(* Logix 5000 project; controller VET 1756-L62 rev 19.52; software revision 19.01; part 12 of 27 *)
(* tags used below, declared in another part *)
   bufferF : REAL[5];
   dosif_struct : ALIAS FOR dosificador[0];
   dosificacion_interrumpida : BOOL;
   dosificando : BOOL;
   falla_struct : falla_aux;
   flags : DINT;
   frq : ALIAS FOR dosif_struct.frq_terreno;
   frq_calculada : REAL;
   idx_batch : DINT;
   idx_bin : DINT;
   idx_ing : DINT;
   idx_tabbin : DINT;
   idx_tolv : DINT;   // Índice de Tolva
   limite_err_inf : REAL;
   limite_err_sup : REAL;
   mensaje : ALIAS FOR dosif_struct.msg;
   peso_delta : REAL;
   peso_detencion : REAL;
   peso_max : REAL;
   peso_medido : ALIAS FOR dosif_struct.peso_terreno;
   peso_neto : REAL;
   peso_objetivo : REAL;
   precorte : REAL;
   respuesta : ALIAS FOR dosif_struct.ans;
   resultado : ALIAS FOR dosif_struct.resultado;
   setD : DINT[5];
   setF : REAL[5];
   step_index : DINT;
   step_index_buffer : DINT;
   T : TIMER[15];
   t_espera : DINT;
   t_pulso : DINT;
   tara : REAL;
   _Eqp : Equipo[800];
   Batch : batch[10];
   Dosificar_MAC_01 : PHASE;
   fecha_plc : DINT;
   hora_plc : DINT;
   TabBin : Bins_Setup;
(* Dosificar_MAC_01, continued *)

ROUTINE dosificar   (* ladder *)
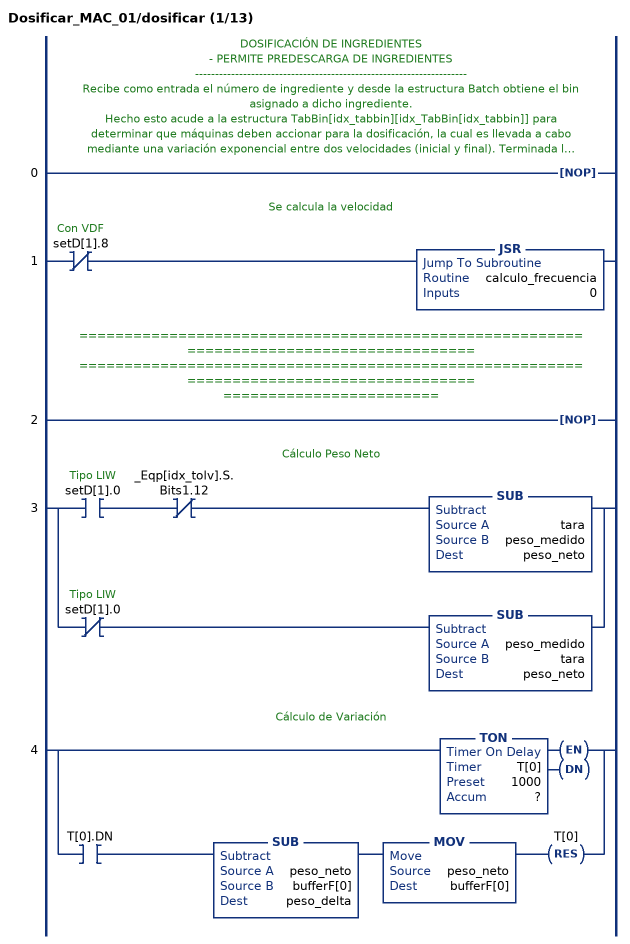
   // DOSIFICACIÓN DE INGREDIENTES
   // - PERMITE PREDESCARGA DE INGREDIENTES
   // --------------------------------------------------------------------
   // Recibe como entrada el número de ingrediente y desde la estructura Batch obtiene el bin asignado a dicho ingrediente.
   // Hecho esto acude a la estructura TabBin[idx_tabbin][idx_TabBin[idx_tabbin]] para determinar que máquinas deben accionar para la dosificación, la cual es llevada a cabo
   // mediante una variación exponencial entre dos velocidades (inicial y final). Terminada la dosificación, se retornan o consolidan los aprendizajes
   // prBatchios de la dosificación, reflejados en un precorte ajustado.
   0: NOP();
   // Se calcula la velocidad
   1: XIO(setD[1].8)JSR(calculo_frecuencia,0);
   // ========================================================================================
   // ========================================================================================
   // ========================
   2: NOP();
   // Cálculo Peso Neto
   3: [XIC(setD[1].0) XIO(_Eqp[idx_tolv].S.Bits1.12) SUB(tara,peso_medido,peso_neto) ,XIO(setD[1].0) SUB(peso_medido,tara,peso_neto) ];
   // Cálculo de Variación
   4: [TON(T[0],?,?) ,XIC(T[0].DN) SUB(peso_neto,bufferF[0],peso_delta) MOV(peso_neto,bufferF[0]) RES(T[0]) ];
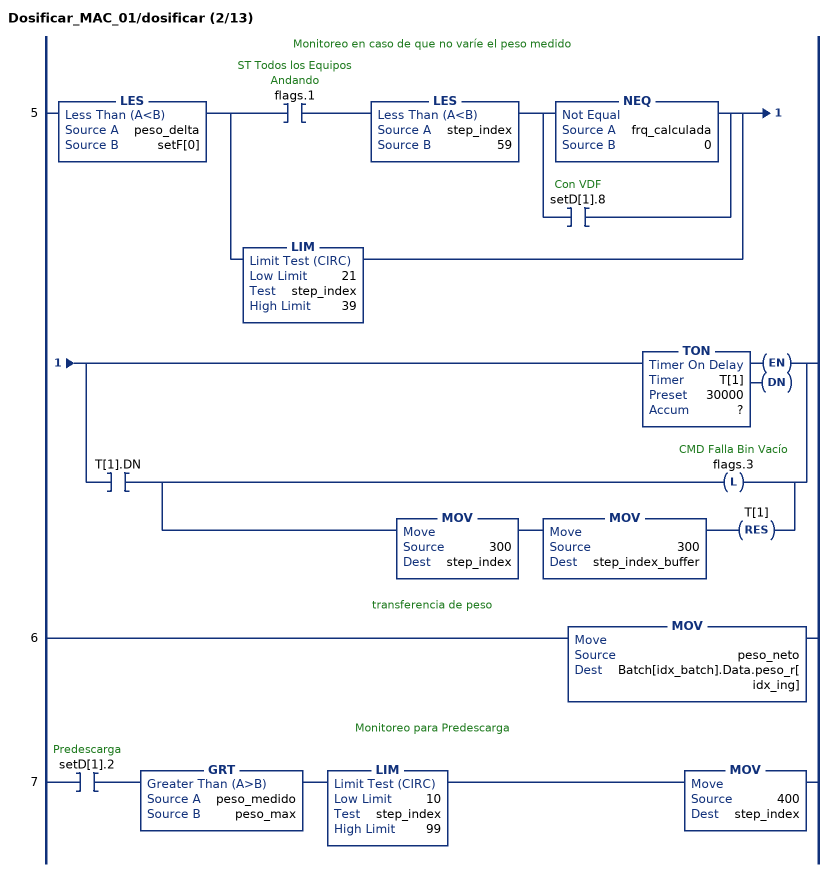
   // Monitoreo en caso de que no varíe el peso medido
   5: LES(peso_delta,setF[0])[XIC(flags.1) LES(step_index,59) [NEQ(frq_calculada,0) ,XIC(setD[1].8) ] ,LIM(21,step_index,39) ][TON(T[1],?,?) ,XIC(T[1].DN) [OTL(flags.3) ,MOV(300,step_index) MOV(300,step_index_buffer) RES(T[1]) ] ];
   // transferencia de peso
   6: MOV(peso_neto,Batch[idx_batch].Data.peso_r[idx_ing]);
   // Monitoreo para Predescarga
   7: XIC(setD[1].2)GRT(peso_medido,peso_max)LIM(10,step_index,99)MOV(400,step_index);
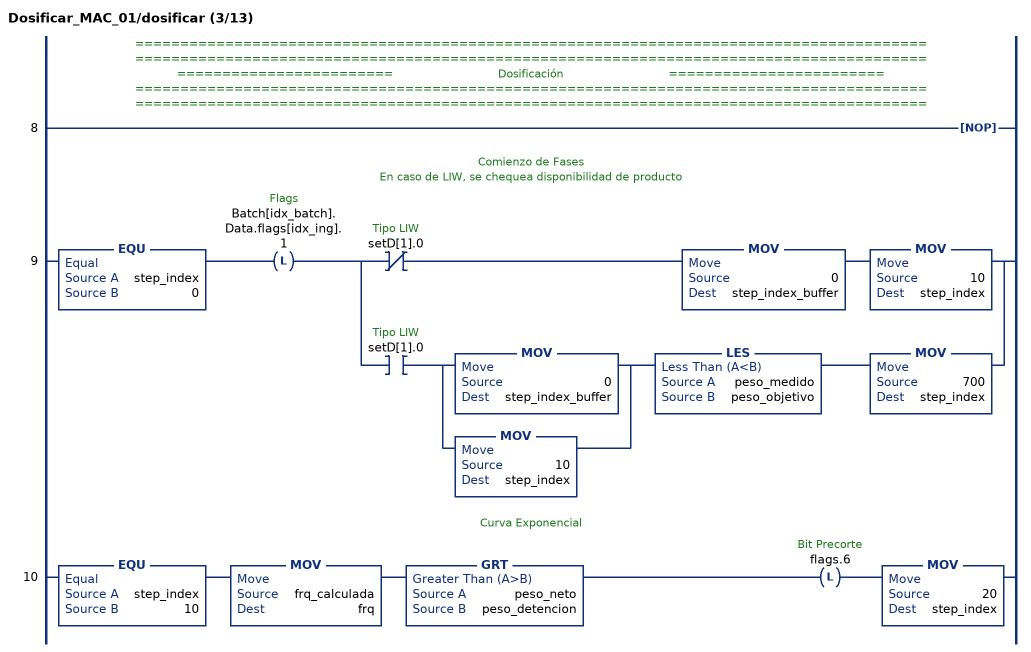
   // ========================================================================================
   // ========================================================================================
   // ========================                              Dosificación                              ========================
   // ========================================================================================
   // ========================================================================================
   8: NOP();
   // Comienzo de Fases
   // En caso de LIW, se chequea disponibilidad de producto
   9: EQU(step_index,0)OTL(Batch[idx_batch].Data.flags[idx_ing].1)[XIO(setD[1].0) MOV(0,step_index_buffer) MOV(10,step_index) ,XIC(setD[1].0) [MOV(0,step_index_buffer) ,MOV(10,step_index) ] LES(peso_medido,peso_objetivo) MOV(700,step_index) ];
   // Curva Exponencial
   10: EQU(step_index,10)MOV(frq_calculada,frq)GRT(peso_neto,peso_detencion)OTL(flags.6)MOV(20,step_index);
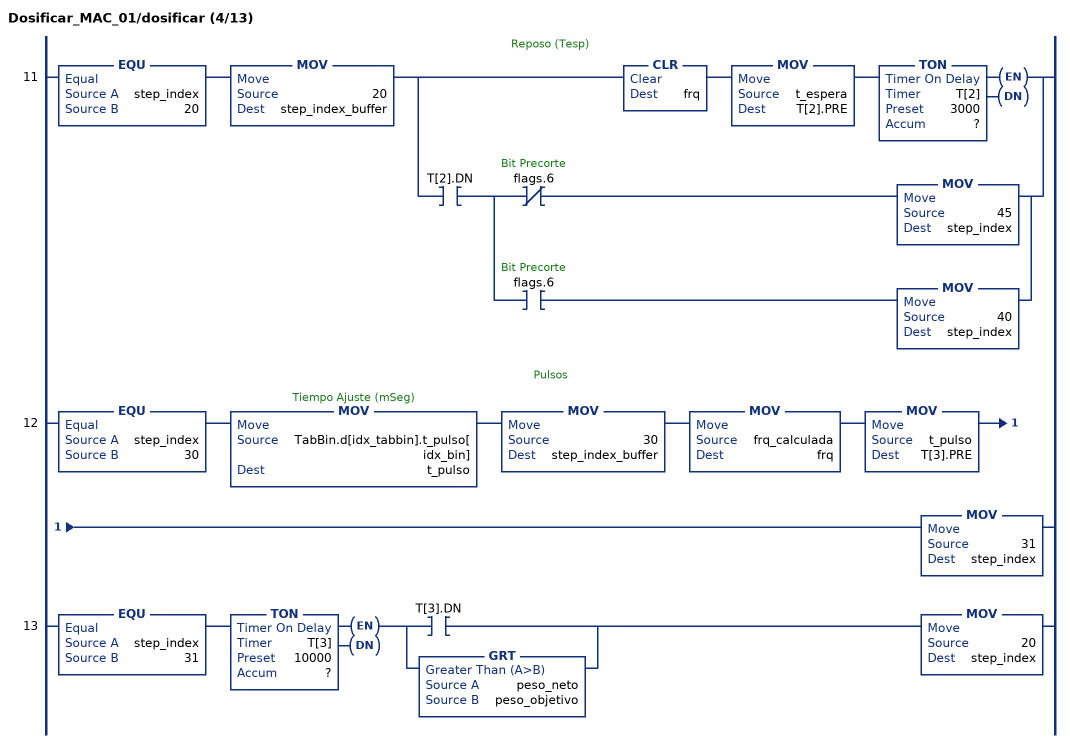
   // Reposo (Tesp)
   11: EQU(step_index,20)MOV(20,step_index_buffer)[CLR(frq) MOV(t_espera,T[2].PRE) TON(T[2],?,?) ,XIC(T[2].DN) [XIO(flags.6) MOV(45,step_index) ,XIC(flags.6) MOV(40,step_index) ] ];
   // Pulsos
   12: EQU(step_index,30)MOV(TabBin.d[idx_tabbin].t_pulso[idx_bin],t_pulso)MOV(30,step_index_buffer)MOV(frq_calculada,frq)MOV(t_pulso,T[3].PRE)MOV(31,step_index);
   13: EQU(step_index,31)TON(T[3],?,?)[XIC(T[3].DN) ,GRT(peso_neto,peso_objetivo) ]MOV(20,step_index);
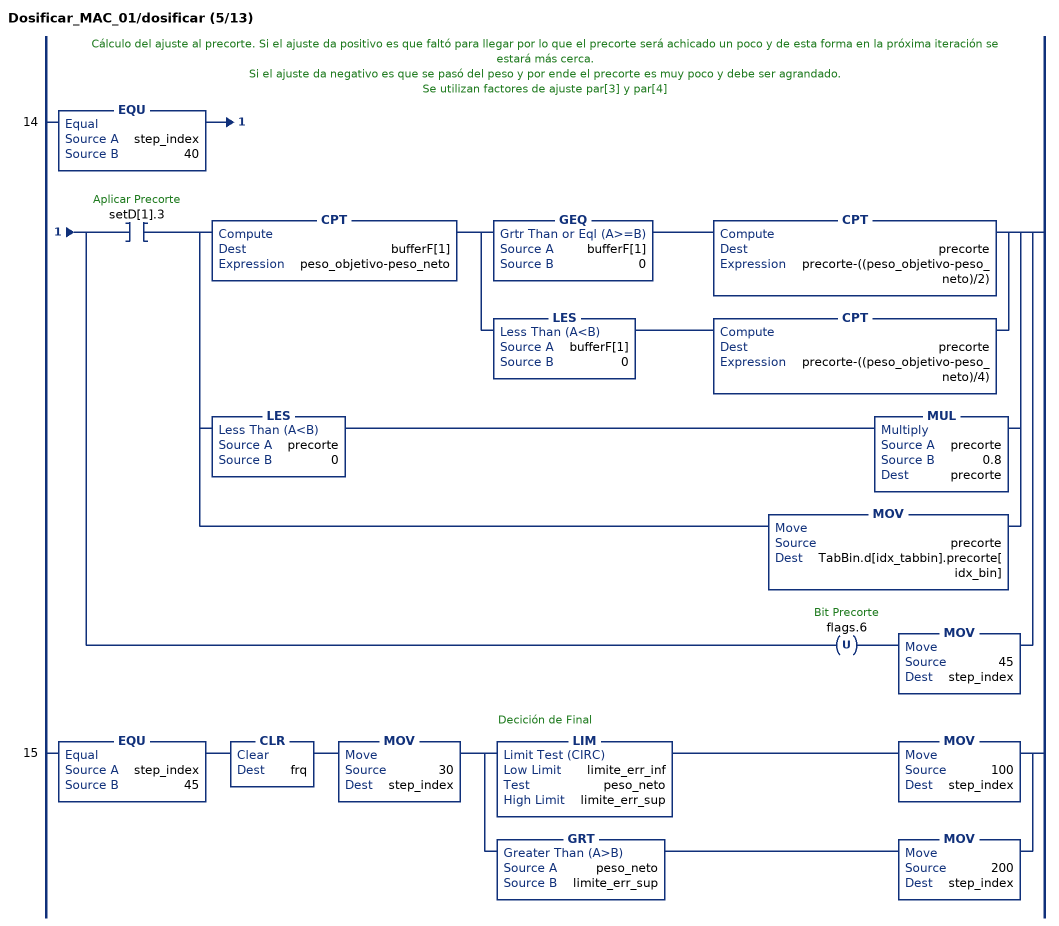
   // Cálculo del ajuste al precorte. Si el ajuste da positivo es que faltó para llegar por lo que el precorte será achicado un poco y de esta forma en la próxima iteración se estará más cerca.
   // Si el ajuste da negativo es que se pasó del peso y por ende el precorte es muy poco y debe ser agrandado.
   // Se utilizan factores de ajuste par[3] y par[4]
   14: EQU(step_index,40)[XIC(setD[1].3) [CPT(bufferF[1],peso_objetivo-peso_neto) [GEQ(bufferF[1],0) CPT(precorte,precorte-((peso_objetivo-peso_neto)/2)) ,LES(bufferF[1],0) CPT(precorte,precorte-((peso_objetivo-peso_neto)/4)) ] ,LES(precorte,0) MUL(precorte,0.8,precorte) ,MOV(precorte,TabBin.d[idx_tabbin].precorte[idx_bin]) ] ,OTU(flags.6) MOV(45,step_index) ];
   // Decición de Final
   15: EQU(step_index,45)CLR(frq)MOV(30,step_index)[LIM(limite_err_inf,peso_neto,limite_err_sup) MOV(100,step_index) ,GRT(peso_neto,limite_err_sup) MOV(200,step_index) ];
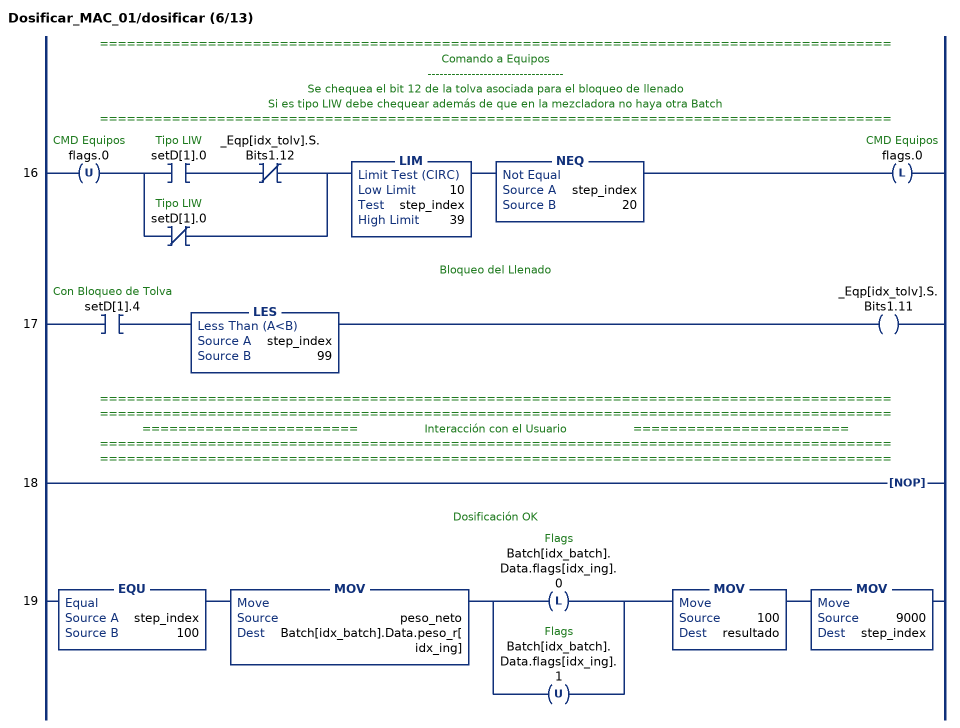
   // ========================================================================================
   // Comando a Equipos
   // ----------------------------------
   // Se chequea el bit 12 de la tolva asociada para el bloqueo de llenado
   // Si es tipo LIW debe chequear además de que en la mezcladora no haya otra Batch
   // ========================================================================================
   16: OTU(flags.0)[XIC(setD[1].0) XIO(_Eqp[idx_tolv].S.Bits1.12) ,XIO(setD[1].0) ]LIM(10,step_index,39)NEQ(step_index,20)OTL(flags.0);
   // Bloqueo del Llenado
   17: XIC(setD[1].4)LES(step_index,99)OTE(_Eqp[idx_tolv].S.Bits1.11);
   // ========================================================================================
   // ========================================================================================
   // ========================                   Interacción con el Usuario                   ========================
   // ========================================================================================
   // ========================================================================================
   18: NOP();
   // Dosificación OK
   19: EQU(step_index,100)MOV(peso_neto,Batch[idx_batch].Data.peso_r[idx_ing])[OTL(Batch[idx_batch].Data.flags[idx_ing].0) ,OTU(Batch[idx_batch].Data.flags[idx_ing].1) ]MOV(100,resultado)MOV(9000,step_index);
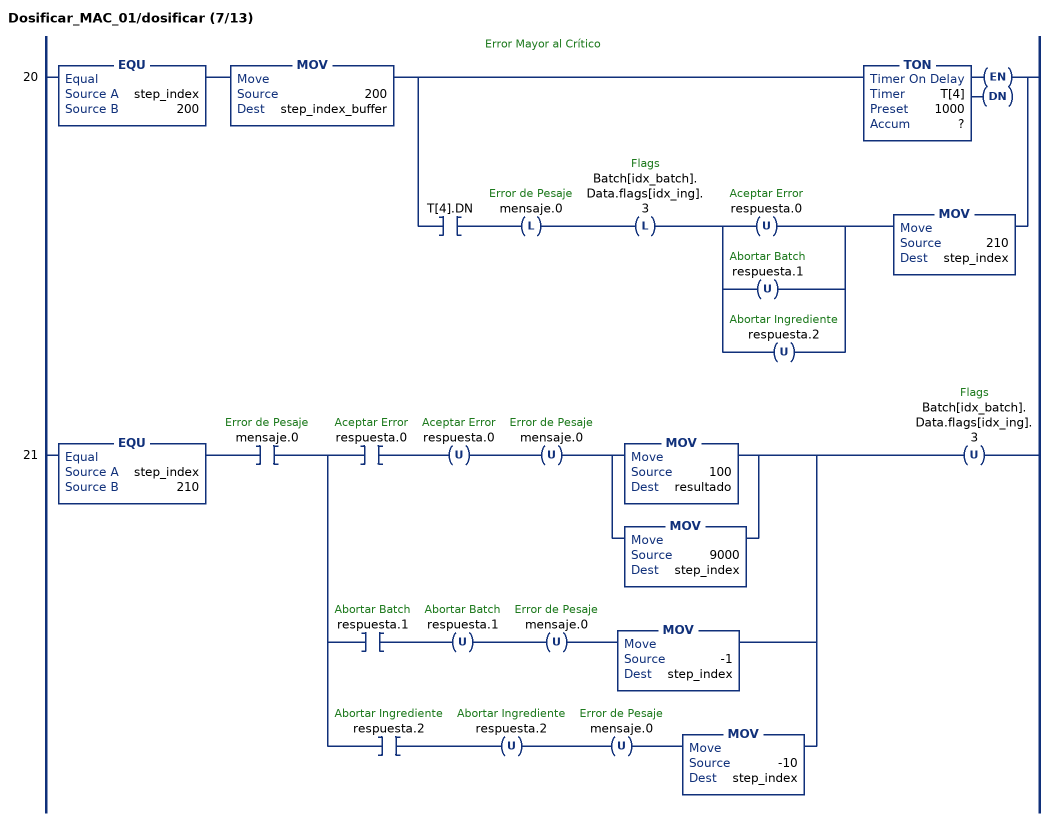
   // Error Mayor al Crítico
   20: EQU(step_index,200)MOV(200,step_index_buffer)[TON(T[4],?,?) ,XIC(T[4].DN) OTL(mensaje.0) OTL(Batch[idx_batch].Data.flags[idx_ing].3) [OTU(respuesta.0) ,OTU(respuesta.1) ,OTU(respuesta.2) ] MOV(210,step_index) ];
   21: EQU(step_index,210)XIC(mensaje.0)[XIC(respuesta.0) OTU(respuesta.0) OTU(mensaje.0) [MOV(100,resultado) ,MOV(9000,step_index) ] ,XIC(respuesta.1) OTU(respuesta.1) OTU(mensaje.0) MOV(-1,step_index) ,XIC(respuesta.2) OTU(respuesta.2) OTU(mensaje.0) MOV(-10,step_index) ]OTU(Batch[idx_batch].Data.flags[idx_ing].3);
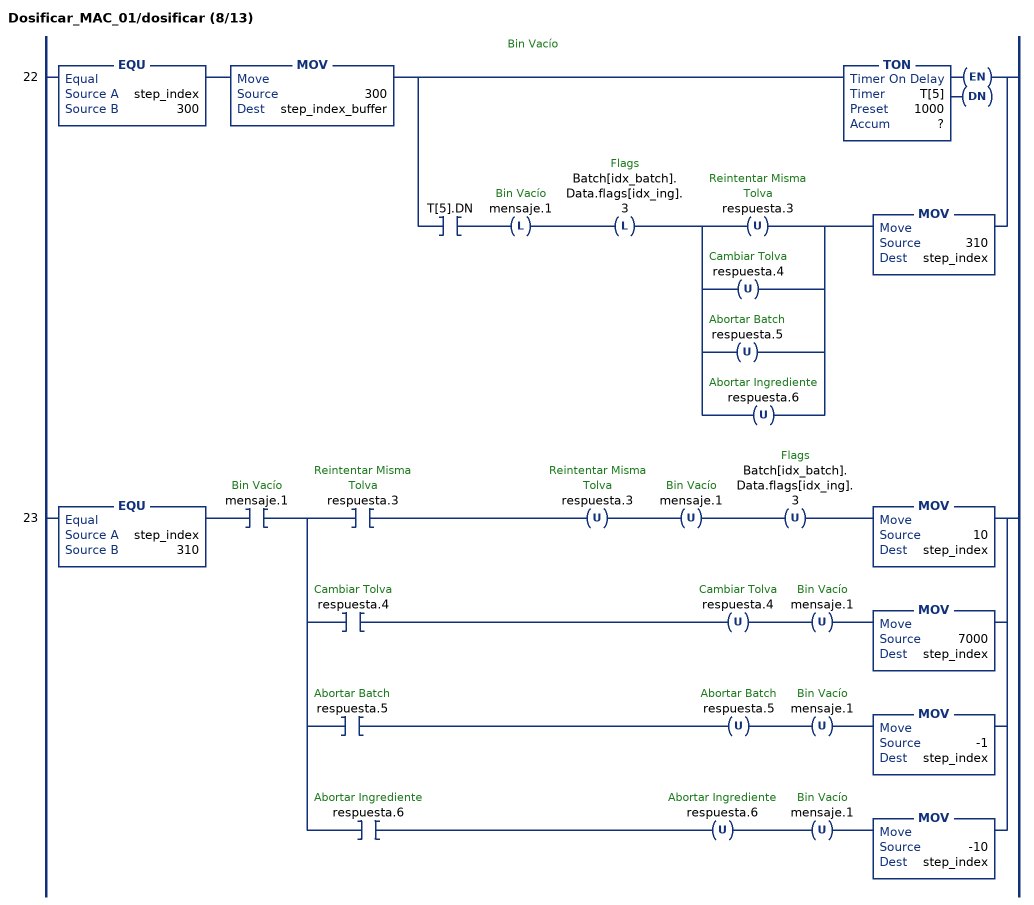
   // Bin Vacío
   22: EQU(step_index,300)MOV(300,step_index_buffer)[TON(T[5],?,?) ,XIC(T[5].DN) OTL(mensaje.1) OTL(Batch[idx_batch].Data.flags[idx_ing].3) [OTU(respuesta.3) ,OTU(respuesta.4) ,OTU(respuesta.5) ,OTU(respuesta.6) ] MOV(310,step_index) ];
   23: EQU(step_index,310)XIC(mensaje.1)[XIC(respuesta.3) OTU(respuesta.3) OTU(mensaje.1) OTU(Batch[idx_batch].Data.flags[idx_ing].3) MOV(10,step_index) ,XIC(respuesta.4) OTU(respuesta.4) OTU(mensaje.1) MOV(7000,step_index) ,XIC(respuesta.5) OTU(respuesta.5) OTU(mensaje.1) MOV(-1,step_index) ,XIC(respuesta.6) OTU(respuesta.6) OTU(mensaje.1) MOV(-10,step_index) ];
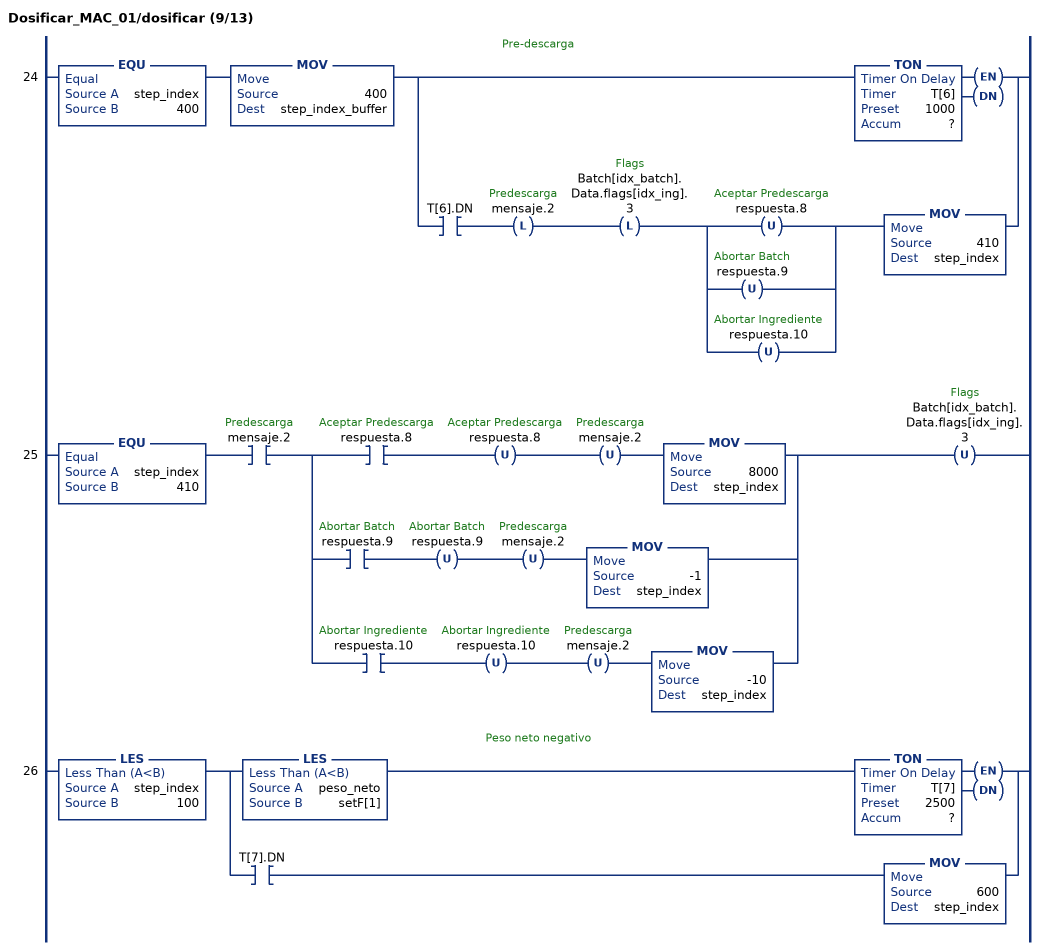
   // Pre-descarga
   24: EQU(step_index,400)MOV(400,step_index_buffer)[TON(T[6],?,?) ,XIC(T[6].DN) OTL(mensaje.2) OTL(Batch[idx_batch].Data.flags[idx_ing].3) [OTU(respuesta.8) ,OTU(respuesta.9) ,OTU(respuesta.10) ] MOV(410,step_index) ];
   25: EQU(step_index,410)XIC(mensaje.2)[XIC(respuesta.8) OTU(respuesta.8) OTU(mensaje.2) MOV(8000,step_index) ,XIC(respuesta.9) OTU(respuesta.9) OTU(mensaje.2) MOV(-1,step_index) ,XIC(respuesta.10) OTU(respuesta.10) OTU(mensaje.2) MOV(-10,step_index) ]OTU(Batch[idx_batch].Data.flags[idx_ing].3);
   // Peso neto negativo
   26: LES(step_index,100)[LES(peso_neto,setF[1]) TON(T[7],?,?) ,XIC(T[7].DN) MOV(600,step_index) ];
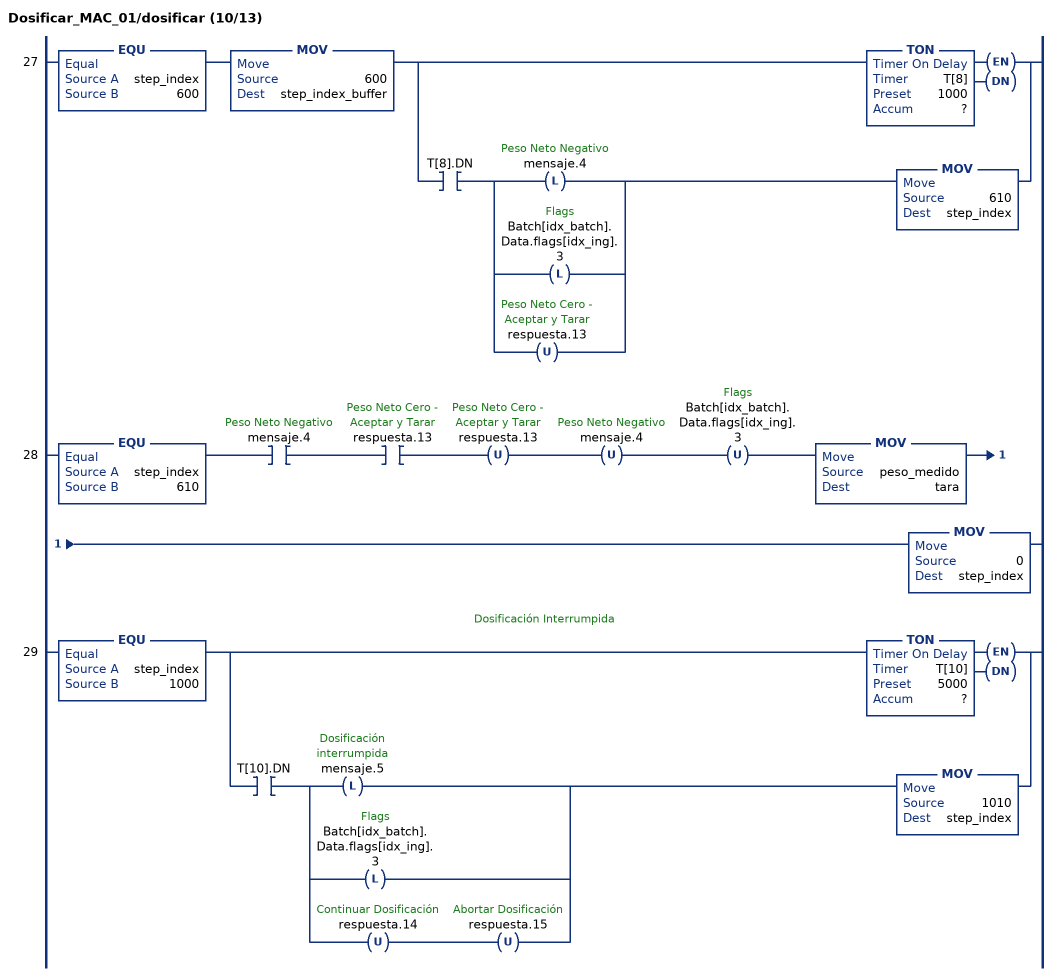
   27: EQU(step_index,600)MOV(600,step_index_buffer)[TON(T[8],?,?) ,XIC(T[8].DN) [OTL(mensaje.4) ,OTL(Batch[idx_batch].Data.flags[idx_ing].3) ,OTU(respuesta.13) ] MOV(610,step_index) ];
   28: EQU(step_index,610)XIC(mensaje.4)XIC(respuesta.13)OTU(respuesta.13)OTU(mensaje.4)OTU(Batch[idx_batch].Data.flags[idx_ing].3)MOV(peso_medido,tara)MOV(0,step_index);
   // Dosificación Interrumpida
   29: EQU(step_index,1000)[TON(T[10],?,?) ,XIC(T[10].DN) [OTL(mensaje.5) ,OTL(Batch[idx_batch].Data.flags[idx_ing].3) ,OTU(respuesta.14) OTU(respuesta.15) ] MOV(1010,step_index) ];
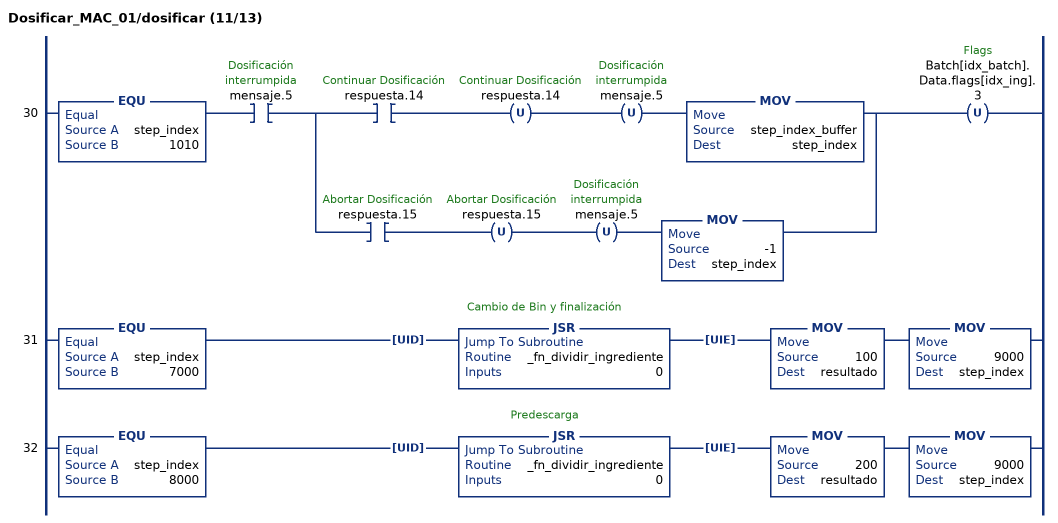
   30: EQU(step_index,1010)XIC(mensaje.5)[XIC(respuesta.14) OTU(respuesta.14) OTU(mensaje.5) MOV(step_index_buffer,step_index) ,XIC(respuesta.15) OTU(respuesta.15) OTU(mensaje.5) MOV(-1,step_index) ]OTU(Batch[idx_batch].Data.flags[idx_ing].3);
   // Cambio de Bin y finalización
   31: EQU(step_index,7000)UID()JSR(_fn_dividir_ingrediente,0)UIE()MOV(100,resultado)MOV(9000,step_index);
   // Predescarga
   32: EQU(step_index,8000)UID()JSR(_fn_dividir_ingrediente,0)UIE()MOV(200,resultado)MOV(9000,step_index);
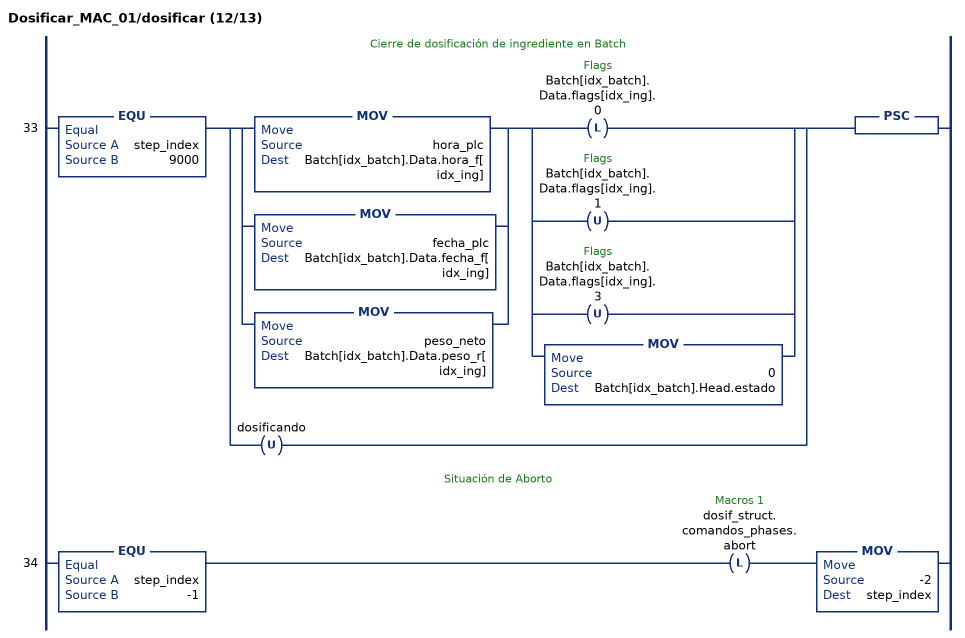
   // Cierre de dosificación de ingrediente en Batch
   33: EQU(step_index,9000)[[MOV(hora_plc,Batch[idx_batch].Data.hora_f[idx_ing]) ,MOV(fecha_plc,Batch[idx_batch].Data.fecha_f[idx_ing]) ,MOV(peso_neto,Batch[idx_batch].Data.peso_r[idx_ing]) ] [OTL(Batch[idx_batch].Data.flags[idx_ing].0) ,OTU(Batch[idx_batch].Data.flags[idx_ing].1) ,OTU(Batch[idx_batch].Data.flags[idx_ing].3) ,MOV(0,Batch[idx_batch].Head.estado) ] ,OTU(dosificando) ]PSC();
   // Situación de Aborto
   34: EQU(step_index,-1)OTL(dosif_struct.comandos_phases.abort)MOV(-2,step_index);
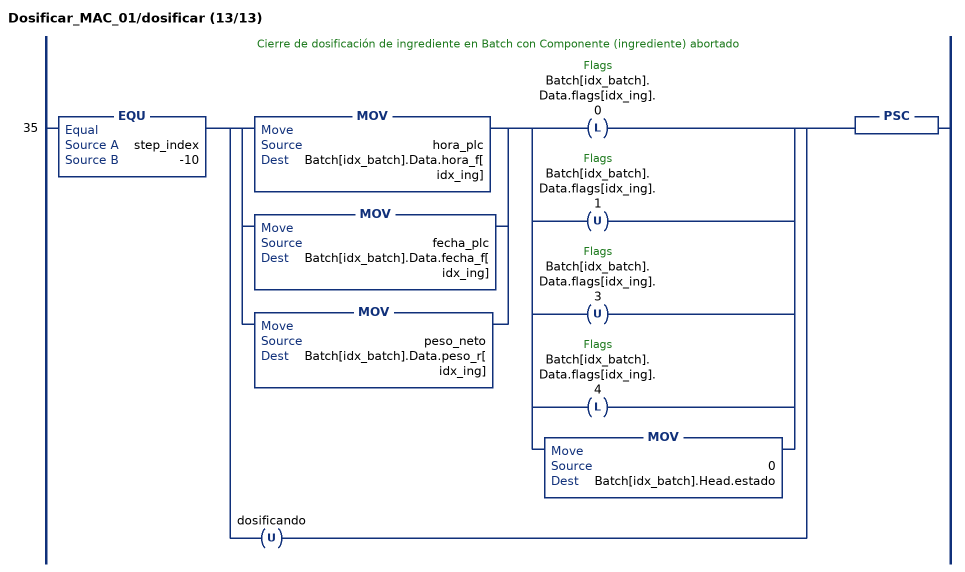
   // Cierre de dosificación de ingrediente en Batch con Componente (ingrediente) abortado
   35: EQU(step_index,-10)[[MOV(hora_plc,Batch[idx_batch].Data.hora_f[idx_ing]) ,MOV(fecha_plc,Batch[idx_batch].Data.fecha_f[idx_ing]) ,MOV(peso_neto,Batch[idx_batch].Data.peso_r[idx_ing]) ] [OTL(Batch[idx_batch].Data.flags[idx_ing].0) ,OTU(Batch[idx_batch].Data.flags[idx_ing].1) ,OTU(Batch[idx_batch].Data.flags[idx_ing].3) ,OTL(Batch[idx_batch].Data.flags[idx_ing].4) ,MOV(0,Batch[idx_batch].Head.estado) ] ,OTU(dosificando) ]PSC();
END_ROUTINE

ROUTINE Falla   (* ladder *)
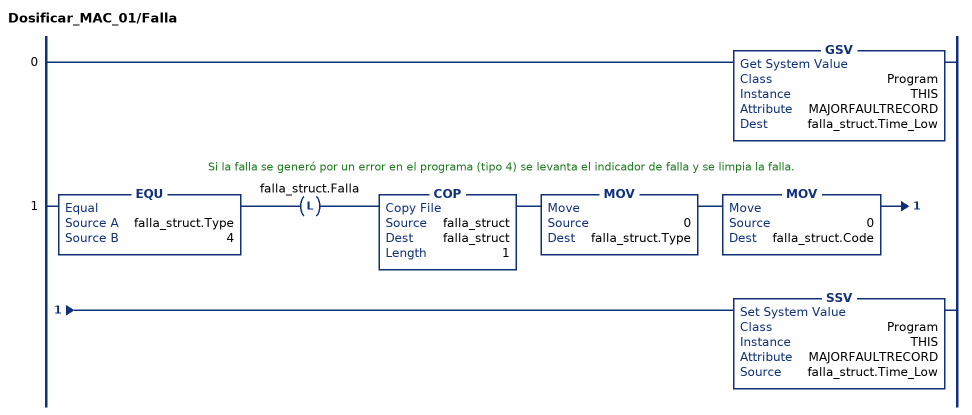
   0: GSV(Program,THIS,MAJORFAULTRECORD,falla_struct.Time_Low);
   // Si la falla se generó por un error en el programa (tipo 4) se levanta el indicador de falla y se limpia la falla.
   1: EQU(falla_struct.Type,4)OTL(falla_struct.Falla)COP(falla_struct,falla_struct,1)MOV(0,falla_struct.Type)MOV(0,falla_struct.Code)SSV(Program,THIS,MAJORFAULTRECORD,falla_struct.Time_Low);
END_ROUTINE

ROUTINE Holding   (* ladder *)
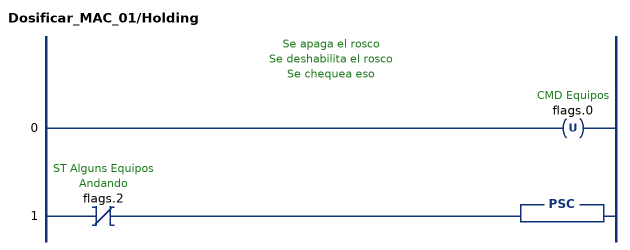
   // Se apaga el rosco
   // Se deshabilita el rosco
   // Se chequea eso
   0: OTU(flags.0);
   1: XIO(flags.2)PSC();
END_ROUTINE

ROUTINE preState   (* ladder *)
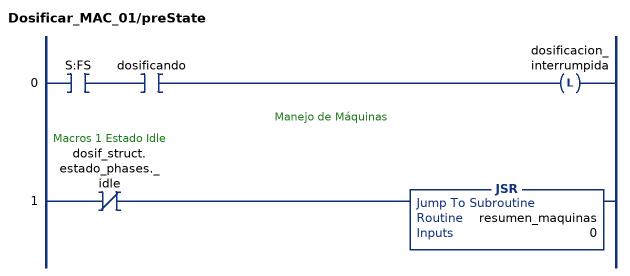
   0: XIC(S:FS)XIC(dosificando)OTL(dosificacion_interrumpida);
   // Manejo de Máquinas
   1: XIO(dosif_struct.estado_phases._idle)JSR(resumen_maquinas,0);
END_ROUTINE

ROUTINE Resetting   (* ladder *)
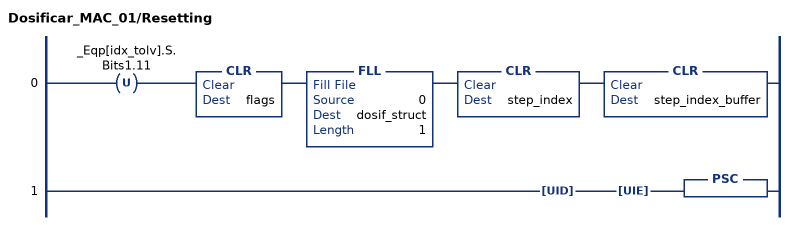
   0: OTU(_Eqp[idx_tolv].S.Bits1.11)CLR(flags)FLL(0,dosif_struct,1)CLR(step_index)CLR(step_index_buffer);
   1: UID()UIE()PSC();
END_ROUTINE

ROUTINE Restarting   (* ladder *)
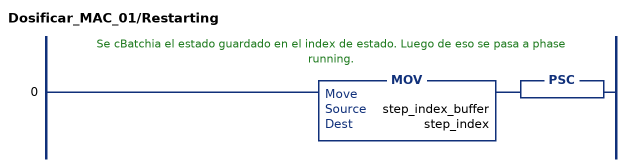
   // Se cBatchia el estado guardado en el index de estado. Luego de eso se pasa a phase running.
   0: MOV(step_index_buffer,step_index)PSC();
END_ROUTINE
